{attribute 'enable_dynamic_creation'}
FUNCTION_BLOCK FB_Cylinder IMPLEMENTS I_Object
VAR_INPUT
END_VAR
VAR_OUTPUT
END_VAR
VAR
	sObjectID			: STRING;
	eObjectType			: E_OBJECTS;
	// pointers for destructor
	_pInstance			: POINTER TO FB_Cylinder;
	_pTemp				: POINTER TO FB_Cylinder;
END_VAR

METHOD Destruct : BOOL
// destroy the instance 
IF _pInstance	<> 0 THEN
	// store in temp value otherwise the FB_exit called at __DELETE will create a stack overflow
	// when not set to 0 before __DELETE  
	_pTemp := _pInstance;
	_pInstance := 16#0; 
	__DELETE(_pTemp);
END_IF
END_METHOD

METHOD FB_init : BOOL
VAR_INPUT
	bInitRetains       : BOOL; // if TRUE, the retain variables are initialized (warm start / cold start)
	bInCopyCode        : BOOL;  // if TRUE, the instance afterwards gets moved into the copy code (online change)
	// Object identifier name
	sObjectID			: STRING;	
	// Object type as a string
	eObjectType			: E_OBJECTS;
END_VAR
THIS^.sObjectID		:= sObjectID;
THIS^.eObjectType	:= eObjectType;
END_METHOD

METHOD M_GetObjectDescription : string
VAR_INPUT
END_VAR
VAR
	sDescription			: STRING;
END_VAR
sDescription := concat(THIS^.sObjectID, ' Type: '); 
sDescription := concat(sDescription, TO_STRING(THIS^.eObjectType)); 
M_GetObjectDescription := sDescription;
END_METHOD

{warning 'add method implementation'}
METHOD M_Reset : BOOL
END_METHOD

{warning 'add method implementation'}
METHOD M_Start : BOOL
END_METHOD

{warning 'add property implementation'}
PROPERTY P_Status : DWORD
GET
END_GET
END_PROPERTY

PROPERTY pInstance : POINTER TO FB_EmptyObject
SET
// Store pointer for destructor
_pInstance := pInstance;
END_SET
END_PROPERTY

END_FUNCTION_BLOCK

(* stored: Version 1.1.0.1, ProductVersion 3.1.4022.18
   POU FB_Cylinder: Id {b732b452-0895-4ab3-bd35-7b01e0123625}, SpecialFunc None
   Method Destruct: Id {509c82fb-3530-44c0-b6b1-172bddbe88c2}
   Method FB_init: Id {a11c6e35-018c-448c-b06a-5448c5cceaf9}
   Method M_GetObjectDescription: Id {294a967c-f617-4f52-a899-d62d471603e2}
   Method M_Reset: Id {70cf5d11-bac3-4e1c-bc4f-da842bbfb5bd}
   Method M_Start: Id {f4e0635b-95a5-4374-a5db-8b46f0d1474b}
   Property P_Status: Id {ca4c5a71-4e68-48bf-8df1-6995bd144bdd}
   Get Get: Id {4b89d285-ad37-4a57-9c6f-3b257a659d89}
   Property pInstance: Id {a355c21f-1afe-473c-af7a-d16ce0b0d882}
   Set Set: Id {4f2b54e3-0fe5-408e-8732-39d3b7ca2849} *)
